IF DSA31ArmSpeedProfileCall.bCallCompleted THEN
DSA31ArmSpeedProfileCall.bCallPB := FALSE;
DSfbGnrProductRecipeMemoryOut.DSGnrCalledArmPnpParameter.DSA1DownPickMovement.lrZone1SpeedVelo := DSA31ArmSpeedProfileCall.Call_DSArmSpdProfile.lrSpeedVelo;
DSfbGnrProductRecipeMemoryOut.DSGnrCalledArmPnpParameter.DSA1DownPickMovement.lrZone1Acc := DSA31ArmSpeedProfileCall.Call_DSArmSpdProfile.lrAcc;
DSfbGnrProductRecipeMemoryOut.DSGnrCalledArmPnpParameter.DSA1DownPickMovement.lrZone1Dcc := DSA31ArmSpeedProfileCall.Call_DSArmSpdProfile.lrDcc;

DSfbGnrProductRecipeMemoryOut.iCallCaseNo:=22;
END_IF

IF rebInvalidSpeedProfileMemoryCall.Q THEN
DSA31ArmSpeedProfileCall.bCallPB := FALSE;

DSfbGnrProductRecipeMemoryOut.iCallCaseNo:=82;
END_IF

(*[][][][][][][][][][][][][][][][][][][][][][][][][][][][][][][][][][][][][][][][][][][][][][][][][][][][][][][][][][][][][][][][][][][][][][][][][][][][][][][][][][][][][][][][][][][][][][][][][][][]*)



14: (* Call UpPickPattern*)
DSA21UpDownPatternCall.Call_iUpDownPatternNo := DSA1fbPnpSequenceMemoryCall.Call_DsPnpSequenceMemory.ARiUpTransferPatternNo[iProductRecipeStepCall];
DSA21UpDownPatternCall.bCallPB := TRUE;


IF DSA21UpDownPatternCall.bCallCompleted THEN
DSA21UpDownPatternCall.bCallPB := FALSE;
DSBufferUpTransferPattern := DSA21UpDownPatternCall.Call_DsUpDownPattern;
DSfbGnrProductRecipeMemoryOut.DSGnrCalledArmPnpParameter.DSA1UpTransferMovement.sUpDownPatternDescription := DSA21UpDownPatternCall.Call_DsUpDownPattern.sDescription;
DSfbGnrProductRecipeMemoryOut.iCallCaseNo:=21;
END_IF

13: (* Call DownTransferPattern*)
DSA21UpDownPatternCall.Call_iUpDownPatternNo := DSA1fbPnpSequenceMemoryCall.Call_DsPnpSequenceMemory.ARiDownTransferPatternNo[iProductRecipeStepCall];
DSA21UpDownPatternCall.bCallPB := TRUE;


IF DSA21UpDownPatternCall.bCallCompleted THEN
DSA21UpDownPatternCall.bCallPB := FALSE;
DSBufferDownTransferPattern := DSA21UpDownPatternCall.Call_DsUpDownPattern;
DSfbGnrProductRecipeMemoryOut.DSGnrCalledArmPnpParameter.DSA1DownTransferMovement.sUpDownPatternDescription := DSA21UpDownPatternCall.Call_DsUpDownPattern.sDescription;
DSfbGnrProductRecipeMemoryOut.iCallCaseNo:=14;
END_IF

IF rebInvalidUpDownPatternMemoryCall.Q THEN
DSA21UpDownPatternCall.bCallPB := FALSE;

DSfbGnrProductRecipeMemoryOut.iCallCaseNo:=81;
END_IF

12: (* Call UpPickPattern*)
DSA21UpDownPatternCall.Call_iUpDownPatternNo := DSA1fbPnpSequenceMemoryCall.Call_DsPnpSequenceMemory.ARiUpPickPatternNo[iProductRecipeStepCall];
DSA21UpDownPatternCall.bCallPB := TRUE;


IF DSA21UpDownPatternCall.bCallCompleted THEN
DSA21UpDownPatternCall.bCallPB := FALSE;
DSBufferUpPickPattern := DSA21UpDownPatternCall.Call_DsUpDownPattern;
DSfbGnrProductRecipeMemoryOut.DSGnrCalledArmPnpParameter.DSA1UpPickMovement.sUpDownPatternDescription := DSA21UpDownPatternCall.Call_DsUpDownPattern.sDescription;
DSfbGnrProductRecipeMemoryOut.iCallCaseNo:=13;
END_IF

IF rebInvalidUpDownPatternMemoryCall.Q THEN
DSA21UpDownPatternCall.bCallPB := FALSE;

DSfbGnrProductRecipeMemoryOut.iCallCaseNo:=81;
END_IF

11: (* Call DownPickPattern*)
DSA21UpDownPatternCall.Call_iUpDownPatternNo := DSA1fbPnpSequenceMemoryCall.Call_DsPnpSequenceMemory.ARiDownPickPatternNo[iProductRecipeStepCall];
DSA21UpDownPatternCall.bCallPB := TRUE;


IF DSA21UpDownPatternCall.bCallCompleted THEN
DSA21UpDownPatternCall.bCallPB := FALSE;
DSBufferDownPickPattern := DSA21UpDownPatternCall.Call_DsUpDownPattern;
DSfbGnrProductRecipeMemoryOut.DSGnrCalledArmPnpParameter.DSA1DownPickMovement.sUpDownPatternDescription := DSA21UpDownPatternCall.Call_DsUpDownPattern.sDescription;
DSfbGnrProductRecipeMemoryOut.iCallCaseNo:=12;
END_IF

IF rebInvalidUpDownPatternMemoryCall.Q THEN
DSA21UpDownPatternCall.bCallPB := FALSE;

DSfbGnrProductRecipeMemoryOut.iCallCaseNo:=81;
END_IF


10: (*Push UpDownPattern to Buffer*)
iBufferPickStationNo := DSA1fbPnpSequenceMemoryCall.Call_DsPnpSequenceMemory.ARiPickStationNo[iProductRecipeStepCall];
iBufferTransferStationNo := DSA1fbPnpSequenceMemoryCall.Call_DsPnpSequenceMemory.ARiTransferStationNo[iProductRecipeStepCall];

iBufferDownPickPatternNo := DSA1fbPnpSequenceMemoryCall.Call_DsPnpSequenceMemory.ARiDownPickPatternNo[iProductRecipeStepCall];
iBufferUpPickPatternNo := DSA1fbPnpSequenceMemoryCall.Call_DsPnpSequenceMemory.ARiUpPickPatternNo[iProductRecipeStepCall];
iBufferDownTransferPatternNo := DSA1fbPnpSequenceMemoryCall.Call_DsPnpSequenceMemory.ARiDownTransferPatternNo[iProductRecipeStepCall];
iBufferUpTransferPatternNo := DSA1fbPnpSequenceMemoryCall.Call_DsPnpSequenceMemory.ARiUpTransferPatternNo[iProductRecipeStepCall];

DSfbGnrProductRecipeMemoryOut.DSGnrCalledArmPnpParameter.iStnSeqRecipeNo := DSA1fbPnpSequenceMemoryCall.Call_DsPnpSequenceMemory.ARiStnSeqRepNo[iProductRecipeStepCall];
DSfbGnrProductRecipeMemoryOut.DSGnrCalledArmPnpParameter.iLdGroupNo := DSA1fbPnpSequenceMemoryCall.Call_DsPnpSequenceMemory.iLdGroupNo;
DSfbGnrProductRecipeMemoryOut.DSGnrCalledArmPnpParameter.iUldGroupNo := DSA1fbPnpSequenceMemoryCall.Call_DsPnpSequenceMemory.iUldGroupNo;


DSfbGnrProductRecipeMemoryOut.sProductRecipeDescription := DSA1fbPnpSequenceMemoryCall.Call_DsPnpSequenceMemory.sDescription;

DSfbGnrProductRecipeMemoryOut.iCallCaseNo:=11;


71: (*Complete Data Called*)

	IF bEnableCallArmNo THEN
	DSfbGnrProductRecipeMemoryOut.DSGnrCalledArmPnpParameter.iCallArmNo := iCallArmNo;
	ELSE
	DSfbGnrProductRecipeMemoryOut.DSGnrCalledArmPnpParameter.iCallArmNo := DSA1fbPnpSequenceMemoryCall.Call_DsPnpSequenceMemory.ARiCallArmNo[iProductRecipeStepCall];
	END_IF

DSfbGnrProductRecipeMemoryOut.bCallCompleted := TRUE;
CallSelfCheckHR := FALSE;
DSfbGnrProductRecipeMemoryOut.iCallCaseNo:=72;

72:; (*Done without error*)

81:
(*iPreviousProcessStep := iCurrentProcessStep;*)
CallSelfCheckHR := FALSE;
DSfbGnrProductRecipeMemoryOut.bCallUpDownPatternMemoryErr := TRUE;
DSfbGnrProductRecipeMemoryOut.iCallCaseNo:=91;

82:
(*iPreviousProcessStep := iCurrentProcessStep;*)
DSfbGnrProductRecipeMemoryOut.bCallArmSpeedProfileMemoryErr := TRUE;
CallSelfCheckHR := FALSE;
DSfbGnrProductRecipeMemoryOut.iCallCaseNo:=92;

83:
(*iPreviousProcessStep := iCurrentProcessStep;*)
DSfbGnrProductRecipeMemoryOut.bCallPickStationNoErr := TRUE;
CallSelfCheckHR := FALSE;
DSfbGnrProductRecipeMemoryOut.iCallCaseNo:=93;

84:
(*iPreviousProcessStep := iCurrentProcessStep;*)
DSfbGnrProductRecipeMemoryOut.bCallTransferStationNoErr := TRUE;
CallSelfCheckHR := FALSE;
DSfbGnrProductRecipeMemoryOut.iCallCaseNo:=94;



91:; (*Found UpDownPatternMemoryError and Task Not Complete *)

92:; (*Found ArmSpeedProfileMemoryErr and Task Not Complete *)

93:; (*Found PickStationNoErr and Task Not Complete *)

94:; (*Found TransferStationNoErr and Task Not Complete *)



END_CASE

END_FUNCTION_BLOCK

(* stored: Version 1.1.0.1, ProductVersion 3.1.4024.12
   POU fbV2_GnrProductRecipeMemory: Id {2fb6ed31-2b2d-4349-a678-c9f3d6c7b5f8}, SpecialFunc None *)
